{attribute 'qualified_only'}
{attribute 'strict'}
TYPE E_MotorState :
(
	Unknown := 0,
	Running := 1,
	Stalled := 2,
	SpeedingUp := 3,
	SpeedingDown := 4,
	Error := -1
);
END_TYPE

(* stored: Version 1.1.0.1, ProductVersion 3.1.4024.12
   DUT E_MotorState: Id {afc44607-2e2c-4f37-b0fe-c76ea867068b} *)
